		tryLogDiagnosticMessage(
			message := message,
			category := TOF_Core.LOG_CATEGORY.ERROR,
			topic1 := TO_WSTRING(ClassName),
			topic2 := "FileHandleResourceManager.executeRelease",
			topic3 := "FileHandleResourceManager.executeRelease.Done"
		);
	ELSE
		TOF_Core.WideStrings.Append255(
			message,
			"File '",
			TO_WSTRING(_FileOpen.sPathName),
			"' closed");

		tryLogDiagnosticMessage(
			message := message,
			category := TOF_Core.LOG_CATEGORY.INFORMATION,
			topic1 := TO_WSTRING(ClassName),
			topic2 := TO_WSTRING(__POUNAME())
		);
	END_IF

END_IF
END_METHOD


//! <param name="bInCopyCode">
//! if TRUE, the exit method is called for exiting an instance that is copied afterwards (online change).
//! </param>

(*!
<summary>Makes a final best-effort close request for a still-acquired file handle.</summary>
<description>
Does not wait for bBusy to clear or inspect the close result. Callers must complete normal release through
cyclic Execute before destroying this manager; this fallback does not guarantee that the file has closed. Does
not create framework exceptions or format diagnostics. The same fallback runs when bInCopyCode is TRUE; this
method implements no handoff of an active handle to a copied instance. Before online change, callers must
finish normal release and resolve any cleanup error. Under that precondition this fallback has no acquired
handle to close. It cannot prepare an active manager for online change or guarantee uninterrupted file I/O.
</description>
*)
METHOD FB_exit : BOOL
VAR_INPUT
	
	bInCopyCode	: BOOL;
END_VAR
IF _FileHandleAcquired THEN
	_FileClose(hFile := _FileOpen.hFile, bExecute := TRUE);
	_FileOpen(bExecute := FALSE);	
END_IF
END_METHOD

(*!
<summary>Provides the native handle associated with the file resource.</summary>
<description>
Use only during the current acquisition; the value alone is not an acquisition guard. Do not close it
independently or retain it across release.
</description>
*)
{attribute 'monitoring' := 'call'}
PROPERTY FINAL FileHandle : UINT
GET
FileHandle := _FileOpen.hFile;
END_GET
END_PROPERTY

(*!
<summary>Provides the manager-owned typed resource for binding file-content tasks.</summary>
<description>
The reference is valid only while this manager is alive. Obtaining it does not acquire or open a file. It
remains a borrowed view across release and reacquisition; use its handle only during the current acquisition.
Do not delete the resource or modify its borrowed path. No ownership is transferred.
</description>
*)
PROPERTY FileHandleResource : REFERENCE TO FileHandleResource
GET
FileHandleResource REF= _FileHandleResource;
END_GET
END_PROPERTY

(*!
<summary>Provides the configured path for the file operation.</summary>
<description>
Configure before acquisition and keep unchanged through release. Assignment copies the path without opening a
file; StartAcquire rejects a missing path.
</description>
*)
{attribute 'monitoring' := 'call'}
PROPERTY FilePath : Tc2_System.T_MaxString
GET
FilePath := _FileOpen.sPathName;
END_GET
SET
_FileOpen.sPathName := FilePath;
END_SET
END_PROPERTY

(*!
<summary>Finishes a pending open during stopping without starting a new open.</summary>
<description>
TRUE means its response has been processed (or none was pending), and acquisition is no longer scheduled.
Preserve a successfully returned handle so the normal release path can close it.
</description>
*)

METHOD INTERNAL FinishPendingAcquire : BOOL
IF _FileOpen.bBusy THEN
	_FileOpen(bExecute := FALSE);

	IF NOT _FileOpen.bBusy AND_THEN NOT _FileOpen.bError AND_THEN _FileOpen.hFile > 0 THEN
		_FileHandleAcquired := TRUE;
	END_IF
END_IF

FinishPendingAcquire := NOT _FileOpen.bBusy;

IF FinishPendingAcquire THEN
	_Acquiring := FALSE;
END_IF
END_METHOD

(*!
<summary>Returns a borrowed resource object owned by this manager.</summary>
<description>
The caller must not delete the returned object. It may be obtained before acquisition and retained while the
manager remains alive, including across release and reacquisition. The object remains valid after release, but
its presence does not mean the resource is acquired. Use the underlying resource only after successful
acquisition and before release begins. Do not reuse a handle saved from an earlier acquisition after release.
</description>
*)
METHOD GetResource : TOF_Core.IObject
GetResource := _FileHandleResource;
END_METHOD

(*!
<summary>Selects native file access and text or binary flags.</summary>
<description>
Use the valid Tc2_System FOPEN_MODE combinations documented by FileContentManager.ModeFlags. Configure before
acquisition and keep unchanged through release; native opening reports incompatible flags.
</description>
*)

{attribute 'monitoring' := 'call'}

PROPERTY ModeFlags : DWORD
GET
ModeFlags := _FileOpen.nMode;
END_GET
SET
_FileOpen.nMode := ModeFlags;
END_SET
END_PROPERTY

(*!
<summary>Provides the library namespace used in diagnostics.</summary>
<description>Returns borrowed read-only namespace storage; do not modify the referenced string.</description>
*)
{attribute 'monitoring' := 'call'}
PROPERTY NamespaceName : REFERENCE TO STRING
GET
NamespaceName REF= CurrentNamespace.Name;
END_GET
END_PROPERTY

(*!
<summary>Selects the native path context for the filesystem request.</summary>
<description>
Passed to native file opening. Configure before acquisition and keep unchanged through release; the setter
does not validate or open a path.
</description>
*)
{attribute 'monitoring' := 'call'}
PROPERTY PathType : Tc2_System.E_OpenPath
GET
PathType := _FileOpen.ePath;
END_GET
SET
_FileOpen.ePath := PathType;
END_SET
END_PROPERTY

(*!
<summary>Reports whether this manager currently retains an acquired handle.</summary>
<description>
FALSE also occurs before acquisition completes and after a failed best-effort close attempt. This bookkeeping
flag is not proof that the native service physically released a resource.
</description>
*)
{attribute 'monitoring' := 'call'}
PROPERTY ResourceAcquired : BOOL
GET
ResourceAcquired := _FileHandleAcquired;
END_GET
END_PROPERTY

(*!
<summary>Reports the size of this concrete instance in bytes.</summary>
*)
{attribute 'monitoring' := 'call'}
PROPERTY SelfSize : ULINT
GET
SelfSize := XSIZEOF(THIS^);
END_GET
END_PROPERTY

(*!
<summary>Requests opening of the configured file on subsequent Execute calls.</summary>
<description>
Call once with no pending operation. An already acquired handle is retained. An empty FilePath raises an
exception before the request is scheduled. Computed diagnostic strings are held in local buffers for the
duration of the receiving call.
</description>
*)
METHOD StartAcquire
VAR
	formattedLogMessage : WSTRING(255);
END_VAR
IF _FileHandleAcquired THEN
	RETURN;
END_IF

IF TOF_Core.Strings.IsNullOrWhiteSpace(stringToCheck := _FileOpen.sPathName) THEN
	TOF_Core.Exceptions.ThrowDataMemberNotSpecified(
		sourceNamespaceName := NamespaceName,
		sourceClassName := ClassName,
		sourcePOUName := __POUNAME(),
		sourcePosition := __POSITION(),
		dataMemberName := 'FilePath'
	);
END_IF

formattedLogMessage := TOF_Core.WideStrings.Concat255("Attempt to open file '", TO_WSTRING(_FileOpen.sPathName), "'");

tryLogDiagnosticMessage(
	message := formattedLogMessage,
	category := TOF_Core.LOG_CATEGORY.INFORMATION,
	topic1 := TO_WSTRING(ClassName),
	topic2 := TO_WSTRING(__POUNAME())
);

_FileClose(bExecute := FALSE);
_FileOpen(bExecute := FALSE);
_Acquiring := TRUE;
END_METHOD

(*!
<summary>Requests best-effort closing on subsequent Execute calls.</summary>
<description>
Acquisition must have completed or been drained by FinishPendingAcquire. Call once; releasing an absent handle
is allowed. Computed diagnostic strings are held in local buffers for the duration of the receiving call.
</description>
*)
METHOD StartRelease
VAR
	formattedLogMessage : WSTRING(255);
END_VAR
formattedLogMessage := TOF_Core.WideStrings.Concat255("Attempt to close file '", TO_WSTRING(_FileOpen.sPathName), "'");

tryLogDiagnosticMessage(
	message := formattedLogMessage,
	category := TOF_Core.LOG_CATEGORY.INFORMATION,
	topic1 := TO_WSTRING(ClassName),
	topic2 := TO_WSTRING(__POUNAME())
);

IF _FileHandleAcquired THEN
	_Releasing := TRUE;
ELSE
	_FileOpen(bExecute := FALSE);
END_IF
END_METHOD

(*!
<summary>Configures the timeout passed to native operation requests.</summary>
<description>
Shared by native open and close. Configure before acquisition and keep unchanged through release. It is not an
overall resource-lifecycle deadline.
</description>
*)
{attribute 'monitoring' := 'call'}
PROPERTY Timeout : TIME
GET
Timeout := _FileOpen.tTimeout;
END_GET
SET
_FileOpen.tTimeout := Timeout;
_FileClose.tTimeout := Timeout;
END_SET
END_PROPERTY

(*!
<summary>Reports an internal message through the configured diagnostic route.</summary>
<description>
Uses the borrowed DiagnosticLogger directly when present; otherwise retains LogManager topics and routing.
Contains destination exceptions without recursive logging. Returns FALSE on observed terminal allocation
failure; prior diagnostic effects are not rolled back and the fatal latch remains set.
</description>
*)
METHOD PRIVATE tryLogDiagnosticMessage : BOOL
VAR_IN_OUT CONSTANT
	message : TOF_Core.ERROR_MESSAGE;
END_VAR
VAR_INPUT
	category : TOF_Core.LOG_CATEGORY;
	topic1 : WSTRING := "";
	topic2 : WSTRING := "";
	topic3 : WSTRING := "";
END_VAR
__TRY

	IF TOF_Core.DynamicMemoryManager.HasAllocationFailed THEN
		RETURN;
	END_IF

	IF _DiagnosticLogger <> 0 THEN
		tryLogDiagnosticMessage := _DiagnosticLogger.TryLogMessage(category := category, message := message);
	ELSE
		tryLogDiagnosticMessage := TOF_Core.LogManager.TryLogMessage(
			category := category,
			message := message,
			topic1 := topic1,
			topic2 := topic2,
			topic3 := topic3
		);
	END_IF

	IF TOF_Core.DynamicMemoryManager.HasAllocationFailed THEN
		tryLogDiagnosticMessage := FALSE;
	END_IF

__CATCH
	// Diagnostic failure must not replace the task lifecycle outcome.
	tryLogDiagnosticMessage := FALSE;
__ENDTRY
END_METHOD

END_FUNCTION_BLOCK

// ---- Tasks/File/FileContent/FileHandleResource.TcPOU
(*
SPDX-FileCopyrightText: © 2026 Oleksandr Tiutyk <trofimich@gmail.com>
SPDX-License-Identifier: MIT
License: https://opensource.org/license/mit
*)

(*!
<summary>Exposes a borrowed view of the native open-file block owned by a resource manager.</summary>
<description>
This object owns neither the native block nor its handle. Keep the referenced FB_FileOpen alive for the entire
use of this view. The getters do not check acquisition: an assigned view is not evidence of an open file. Use
handle and target together only during the current acquisition, never after release. An invalid native-block
reference yields default scalar results or an invalid FilePath reference. Do not modify FilePath through its
reference, close the handle independently or delete this borrowed object.
</description>
*)

{attribute 'no_explicit_call' := 'Direct call is not allowed'}
FUNCTION_BLOCK INTERNAL FileHandleResource EXTENDS TOF_Core.Object
VAR_STAT
	//! <summary>Class name shared by all instances of this function block.</summary>
	{attribute 'hide'} 
	_ClassName : STRING := __POUNAME();
END_VAR
VAR
	{attribute 'hide'} 
	_FileOpen : REFERENCE TO Tc2_System.FB_FileOpen;
END_VAR

(*!
<summary>Target of the open file; use together with FileHandle.</summary>
*)

{attribute 'monitoring' := 'call'}

PROPERTY AmsNetId : Tc2_System.T_AmsNetID
GET
IF __ISVALIDREF(_FileOpen) THEN
	AmsNetId := _FileOpen.sNetId;
END_IF
END_GET
END_PROPERTY

(*!
<summary>Provides the concrete type name used in diagnostics.</summary>
<description>
Returns borrowed read-only metadata; keep the instance alive and do not modify the referenced string.
Reading does not allocate memory, initialize resources or transfer ownership.
</description>
*)
{attribute 'monitoring' := 'call'}
PROPERTY ClassName : REFERENCE TO STRING
GET
ClassName REF= _ClassName;
END_GET
END_PROPERTY

(*!
<summary>Binds this view to a caller-owned native file-open block without acquiring a file.</summary>
<description>
The binding is borrowed and must remain alive throughout use. An invalid reference is retained without
throwing; getters then return default scalars or an invalid reference. No handle is opened or closed.
</description>
<param name="fileOpen">Borrowed native block providing the path, target and current handle.</param>
*)
METHOD FB_Init: BOOL
VAR_INPUT
	bInitRetains : BOOL; // TRUE: the retain variables are initialized (reset warm / reset cold)
	bInCopyCode : BOOL;  // TRUE: the instance will be copied to the copy code afterward (online change)
	fileOpen : REFERENCE TO Tc2_System.FB_FileOpen;
END_VAR
_FileOpen REF= fileOpen;
END_METHOD

(*!
<summary>Reads the native handle from the borrowed open-file block.</summary>
<description>
Returns the default UINT when no native block is bound. Does not check acquisition or close status; a stored
numeric handle must not be reused after release.
</description>
*)
{attribute 'monitoring' := 'call'}
PROPERTY FileHandle : UINT
GET
IF __ISVALIDREF(_FileOpen) THEN
	FileHandle := _FileOpen.hFile;
END_IF
END_GET
END_PROPERTY

(*!
<summary>Provides a borrowed view of the configured native file path.</summary>
<description>
The reference is invalid when no native block is bound. Keep the owner alive and do not write through this
reference. This path identifies configuration, not proof that the file is open.
</description>
*)
{attribute 'monitoring' := 'call'}
PROPERTY FilePath : REFERENCE TO Tc2_System.T_MaxString
GET
IF __ISVALIDREF(_FileOpen) THEN
	FilePath REF= _FileOpen.sPathName;
END_IF
END_GET
END_PROPERTY

(*!
<summary>Provides the library namespace used in diagnostics.</summary>
<description>Returns borrowed read-only namespace storage; do not modify the referenced string.</description>
*)
{attribute 'monitoring' := 'call'}
PROPERTY NamespaceName : REFERENCE TO STRING
GET
NamespaceName REF= CurrentNamespace.Name;
END_GET
END_PROPERTY

(*!
<summary>Reports the size of this concrete instance in bytes.</summary>
*)
{attribute 'monitoring' := 'call'}
PROPERTY SelfSize : ULINT
GET
SelfSize := XSIZEOF(THIS^);
END_GET
END_PROPERTY

END_FUNCTION_BLOCK

// ---- Tasks/File/FileContent/Tasks/CheckEndOfFile.TcPOU
(*
SPDX-FileCopyrightText: © 2026 Oleksandr Tiutyk <trofimich@gmail.com>
SPDX-License-Identifier: MIT
License: https://opensource.org/license/mit
*)

(*!
<summary>Queries the native end-of-file status of the acquired file.</summary>
<description>
The owner must keep the resource acquired through stopping. Configure Timeout before Start and keep it
unchanged until STOPPED. Missing binding and native errors use the Task failure and cleanup path. IsEndOfFile
exposes the native result only after STOPPED with WORK_DONE; FALSE outside that state does not establish that
more data is available. Cancellation waits for a submitted query. Reset clears binding and request state while
retaining Timeout.
</description>
*)

{attribute 'no_explicit_call' := 'do not call this function block directly'}
FUNCTION_BLOCK CheckEndOfFile EXTENDS FileContentTask
VAR_STAT
	//! <summary>Static type metadata available before the base task initializes its default name.</summary>
	{attribute 'hide'}
	_ClassName : STRING := __POUNAME();
END_VAR
VAR
    _CheckEOF : Tc2_System.FB_EOF;
END_VAR

(*!
<summary>Exposes the native operation target copied from the bound file resource.</summary>
<description>
The resource target overwrites a separately assigned value before native submission. Configure the resource
owner to select a target; do not change this value while the task is running.
</description>
*)
{attribute 'monitoring' := 'call'}
PROPERTY AmsNetId : Tc2_System.T_AmsNetID
GET
AmsNetId := _CheckEOF.sNetId;
END_GET
SET
_CheckEOF.sNetId := AmsNetId;
END_SET
END_PROPERTY

(*!
<summary>Provides the concrete type name used in diagnostics.</summary>
<description>
Returns borrowed read-only metadata; keep the instance alive and do not modify the referenced string.
Initialized static storage is ready during base Task.FB_init; this getter has no side effects or exceptions.
</description>
*)
{attribute 'monitoring' := 'call'}
PROPERTY ClassName : REFERENCE TO STRING
GET
ClassName REF= _ClassName;
END_GET
END_PROPERTY

(*!
<summary>Reports whether the underlying native file operation is busy.</summary>
<description>
Observes native I/O, including work drained during stopping. FALSE is not a task-success result and does not
independently permit the resource owner to close or destroy the file.
</description>
*)
{attribute 'monitoring' := 'call'}
PROPERTY FileOperationInProgress : BOOL
GET
FileOperationInProgress := _CheckEOF.bBusy;
END_GET
END_PROPERTY

(*!
<summary>Reports the EOF indicator obtained by a successfully completed check.</summary>
<description>
Returns the native result only while State.Stopped and FinalStopReason.WorkDone are both TRUE. In every other
state, including READY, RUNNING, failure and cancellation, returns the initial value of the property type.
This default is not a success indicator; inspect the task state and final reason. FALSE outside successful
completion does not establish that more data is available. The getter does not modify native outputs or
buffers. Copy a successful result before Reset or reuse.
</description>
*)
{attribute 'monitoring' := 'call'}
PROPERTY IsEndOfFile : BOOL
GET
IF NOT State.Stopped OR_ELSE NOT FinalStopReason.WorkDone THEN
	RETURN;
END_IF

IsEndOfFile := _CheckEOF.bEOF;
END_GET
END_PROPERTY

(*!
<summary>Provides the library namespace used in diagnostics.</summary>
<description>Returns borrowed read-only namespace storage; do not modify the referenced string.</description>
*)
{attribute 'monitoring' := 'call'}
PROPERTY NamespaceName : REFERENCE TO STRING
GET
NamespaceName REF= CurrentNamespace.Name;
END_GET
END_PROPERTY

(*!
<summary>Resets the native request edge after the task has stopped.</summary>
<description>
Also preserves the inherited resource-binding cleanup. Configured inputs remain available for reuse; borrowed
buffers are not freed or cleared. Pending I/O must finish during stopping before this hook runs.
</description>
*)
METHOD PROTECTED OnReset
SUPER^.OnReset();

_CheckEOF(bExecute := FALSE);
END_METHOD

(*!
<summary>Checks the end-of-file indicator through the bound file handle.</summary>
<description>
Requires a live bound resource whose owner keeps the handle acquired until stopping completes. Native errors
raise an exception for the base Task failure and cleanup path without dynamic string-builder allocations;
completed I/O effects are not rolled back.
</description>
<param name="processingState">BUSY while pending; DONE after native completion without an error.</param>
<param name="stopReasonMessage">Not changed; native failures use exceptions.</param>
*)
METHOD PROTECTED OnRunning
VAR_OUTPUT
	processingState : TOF_Tasks.TASK_PROCESSING_STATE;
END_VAR
VAR_IN_OUT
	stopReasonMessage : TOF_Core.ERROR_MESSAGE;
END_VAR
VAR
	errorMessage : TOF_Core.ERROR_MESSAGE;
END_VAR
IF NOT _CheckEOF.bExecute THEN 
	IF NOT __ISVALIDREF(_FileHandleResource) THEN
		TOF_Core.Exceptions.ThrowDataMemberNotSpecified(
			sourceNamespaceName := NamespaceName,
			sourceClassName := ClassName,
			sourcePOUName := __POUNAME(),
			sourcePosition := __POSITION(),
			dataMemberName := 'FileHandleResource'
		);		
	END_IF
	
	_CheckEOF.sNetId := _FileHandleResource.AmsNetId;
	_CheckEOF.hFile := _FileHandleResource.FileHandle;
END_IF

_CheckEOF(bExecute := TRUE);

IF _CheckEOF.bError THEN
	TOF_Core.WideStrings.Append255(
		errorMessage,
		"An error occurred while checking end of file '",
		TO_WSTRING(FilePath),
		"'");

	FileSystemExceptions.ThrowFileSystem(
		sourceNamespaceName := NamespaceName,
		sourceClassName := ClassName,
		sourcePOUName := __POUNAME(),
		sourcePosition := __POSITION(),
		message := errorMessage,
		errorCode := _CheckEOF.nErrId
	);
END_IF

IF NOT _CheckEOF.bBusy THEN
	processingState := TOF_Tasks.TASK_PROCESSING_STATE.DONE;
END_IF
END_METHOD

(*!
<summary>Wait for an already submitted file operation before allowing handle release.</summary>
<description>
FALSE on bExecute only avoids a new request; it does not abort the pending one. Runs for every stop reason. If
no operation is busy, stopping is ready immediately.
</description>
<param name="readyToRelease">TRUE after pending work has completed and release may begin.</param>
*)

METHOD PROTECTED OnStopping
VAR_OUTPUT
	readyToRelease : BOOL;
END_VAR
IF _CheckEOF.bBusy THEN
	_CheckEOF(bExecute := FALSE);
END_IF

readyToRelease := NOT _CheckEOF.bBusy;
END_METHOD

(*!
<summary>Reports the size of this concrete instance in bytes.</summary>
*)
{attribute 'monitoring' := 'call'}
PROPERTY SelfSize : ULINT
GET
SelfSize := XSIZEOF(THIS^);
END_GET
END_PROPERTY

(*!
<summary>Configures the timeout passed to native operation requests.</summary>
<description>
Set before Start and keep unchanged until STOPPED. Reset preserves this value. It is not an overall task
deadline or a guarantee of resource release after a timeout.
</description>
*)
{attribute 'monitoring' := 'call'}
PROPERTY Timeout : TIME
GET
Timeout := _CheckEOF.tTimeout;
END_GET
SET
_CheckEOF.tTimeout := Timeout;
END_SET
END_PROPERTY

END_FUNCTION_BLOCK

// ---- Tasks/File/FileContent/Tasks/FileContentTask.TcPOU
(*
SPDX-FileCopyrightText: © 2026 Oleksandr Tiutyk <trofimich@gmail.com>
SPDX-License-Identifier: MIT
License: https://opensource.org/license/mit
*)

(*!
<summary>Base for a file-content operation borrowing a manager-owned file resource.</summary>
<description>
Queue membership and resource binding do not transfer ownership. One owner drives the task. Keep the resource
owner alive while using its binding; an assigned reference alone does not prove acquisition. The manager
acquires the file before child execution and waits for child stopping before release. Removing a child from a
queue does not clear the binding. Reset from STOPPED clears it; READY Reset is a no-op. A removed READY child
must explicitly clear or replace its binding before the old owner is destroyed. Descendants overriding OnReset
must preserve binding cleanup. Descendants must finish native pending I/O during stopping before allowing the
parent to release the resource. Do not mutate borrowed resource data.
</description>
*)

FUNCTION_BLOCK ABSTRACT FileContentTask EXTENDS TOF_Tasks.Task IMPLEMENTS IFileContentTask
VAR
	_FileHandleResource : REFERENCE TO FileHandleResource;
END_VAR

(*!
<summary>File-content operations take the actual target from the bound resource</summary>
<description>
before submitting I/O, overriding any separately configured AmsNetId.
</description>
*)

{attribute 'monitoring' := 'call'}

PROPERTY ABSTRACT AmsNetId : Tc2_System.T_AmsNetID
GET
END_GET
SET
END_SET
END_PROPERTY

(*!
<summary>Reads the handle through the current borrowed resource binding.</summary>
<description>
Returns the default UINT when unbound. Does not establish acquisition; use only while the owning manager has
acquired the current file, and do not cache across release.
</description>
*)
{attribute 'monitoring' := 'call'}
PROPERTY FINAL FileHandle : UINT
GET
IF __ISVALIDREF(_FileHandleResource) THEN
	FileHandle := _FileHandleResource.FileHandle;
END_IF
END_GET
END_PROPERTY

(*!
<summary>Exposes the borrowed resource binding for this operation.</summary>
<description>
Returns an invalid reference when unbound. The owner must remain alive throughout access; an assigned
reference does not mean the file is acquired. Do not mutate borrowed data or close the handle independently.
</description>
*)
{attribute 'monitoring' := 'call'}
PROPERTY FINAL FileHandleResource : REFERENCE TO FileHandleResource
GET
IF __ISVALIDREF(_FileHandleResource) THEN
	FileHandleResource REF= _FileHandleResource;
END_IF
END_GET
END_PROPERTY

(*!
<summary>Copies the file path from the current resource binding.</summary>
<description>
Returns the default empty string when unbound. Reading requires the resource owner to remain alive; the path
is configuration and does not prove acquisition.
</description>
*)
{attribute 'monitoring' := 'call'}
PROPERTY FINAL FilePath : Tc2_System.T_MaxString
GET
IF __ISVALIDREF(_FileHandleResource) THEN
	FilePath := _FileHandleResource.FilePath;
END_IF
END_GET
END_PROPERTY

(*!
<summary>Clears the borrowed resource binding when a STOPPED child is reset.</summary>
<description>
Base Reset does not call this hook in READY. Overriding descendants must preserve this cleanup; it neither
closes the file nor removes the task from any queue.
</description>
*)
METHOD PROTECTED OnReset
_FileHandleResource REF= 0;
END_METHOD

(*!
<summary>Bind, replace or clear a borrowed resource only in READY; otherwise throw.</summary>
<description>
An invalid reference clears the binding. Reset a STOPPED task before rebinding. The caller must first remove
the task from any queue; READY alone does not mean it is unqueued. The resource owner must outlive its use by
this task. Queue removal does not clear this binding; READY Reset is a no-op. Clear or replace the binding
explicitly for a removed READY task before destroying the old resource owner.
</description>
*)

METHOD SetFileHandleResource
VAR_INPUT
	fileHandleResource : REFERENCE TO FileHandleResource;
END_VAR
IF NOT State.Ready THEN
	TOF_Core.Exceptions.ThrowStandard(
		sourceNamespaceName := NamespaceName,
		sourceClassName := ClassName,
		sourcePOUName := __POUNAME(),
		sourcePosition := __POSITION(),
		message := "FileHandleResource can only be assigned in READY state"
	);
END_IF

IF __ISVALIDREF(fileHandleResource) THEN
	_FileHandleResource REF= fileHandleResource;
ELSE
	_FileHandleResource REF= 0;
END_IF
END_METHOD

(*!
<summary>Configures the timeout passed to native operation requests.</summary>
<description>
Implementations apply this value to their native requests. Configure before execution and keep stable through
stopping; it is not a deadline for the entire task lifecycle.
</description>
*)
{attribute 'monitoring' := 'call'}
{attribute 'OPC.UA.DA.Property' := '1'}
{attribute 'OPC.UA.DA' := '1'}
PROPERTY ABSTRACT Timeout : TIME
GET
END_GET
SET
END_SET
END_PROPERTY

(*!
<summary>TRUE while the underlying file FB reports a pending request, including</summary>
<description>
cancellation wait. Reading has no side effects and does not indicate task lifecycle state or permission to
release the file resource.
</description>
*)

{attribute 'monitoring' := 'call'}

PROPERTY ABSTRACT FileOperationInProgress : BOOL
GET
END_GET
END_PROPERTY

END_FUNCTION_BLOCK

// ---- Tasks/File/FileContent/Tasks/SetPositionInFile.TcPOU
(*
SPDX-FileCopyrightText: © 2026 Oleksandr Tiutyk <trofimich@gmail.com>
SPDX-License-Identifier: MIT
License: https://opensource.org/license/mit
*)

(*!
<summary>Changes the bound file's position using a configured offset and origin.</summary>
<description>
The resource owner must keep the file acquired through task stopping. Configure Position, Origin and Timeout
before Start and keep them unchanged until STOPPED. Missing binding and native errors use the base Task
failure and cleanup path. Cancellation waits for submitted I/O and does not restore the previous file
position. Reset from STOPPED clears the binding and native request state, preserving offset, origin and
timeout.
</description>
*)

{attribute 'no_explicit_call' := 'do not call this function block directly'}
FUNCTION_BLOCK SetPositionInFile EXTENDS FileContentTask
VAR_STAT
	//! <summary>Static type metadata available before the base task initializes its default name.</summary>
	{attribute 'hide'}
	_ClassName : STRING := __POUNAME();
END_VAR
VAR
    _SetPosition : Tc2_System.FB_FileSeek;
END_VAR

(*!
<summary>Exposes the native operation target copied from the bound file resource.</summary>
<description>
The resource target overwrites a separately assigned value before native submission. Configure the resource
owner to select a target; do not change this value while the task is running.
</description>
*)
{attribute 'monitoring' := 'call'}
PROPERTY AmsNetId : Tc2_System.T_AmsNetID
GET
AmsNetId := _SetPosition.sNetId;
END_GET
SET
_SetPosition.sNetId := AmsNetId;
END_SET
END_PROPERTY

(*!
<summary>Provides the concrete type name used in diagnostics.</summary>
<description>
Returns borrowed read-only metadata; keep the instance alive and do not modify the referenced string.
Initialized static storage is ready during base Task.FB_init; this getter has no side effects or exceptions.
</description>
*)
{attribute 'monitoring' := 'call'}
PROPERTY ClassName : REFERENCE TO STRING
GET
ClassName REF= _ClassName;
END_GET
END_PROPERTY

(*!
<summary>Reports whether the underlying native file operation is busy.</summary>
<description>
Observes native I/O, including work drained during stopping. FALSE is not a task-success result and does not
independently permit the resource owner to close or destroy the file.
</description>
*)
{attribute 'monitoring' := 'call'}
PROPERTY FileOperationInProgress : BOOL
GET
FileOperationInProgress := _SetPosition.bBusy;
END_GET
END_PROPERTY

(*!
<summary>Provides the library namespace used in diagnostics.</summary>
<description>Returns borrowed read-only namespace storage; do not modify the referenced string.</description>
*)
{attribute 'monitoring' := 'call'}
PROPERTY NamespaceName : REFERENCE TO STRING
GET
NamespaceName REF= CurrentNamespace.Name;
END_GET
END_PROPERTY

(*!
<summary>Clears the borrowed binding and native request state after stopping.</summary>
<description>
Preserves Position, Origin and Timeout. Does not cancel pending I/O; stopping must finish first.
</description>
*)
METHOD PROTECTED OnReset
SUPER^.OnReset();

_SetPosition(bExecute := FALSE);
END_METHOD

(*!
<summary>Changes the position of the bound file using the configured offset and origin.</summary>
<description>
Requires a live bound resource whose owner keeps the handle acquired until stopping completes. Native errors
raise an exception for the base Task failure and cleanup path without dynamic string-builder allocations;
completed I/O effects are not rolled back.
</description>
<param name="processingState">BUSY while pending; DONE after native completion without an error.</param>
<param name="stopReasonMessage">Not changed; native failures use exceptions.</param>
*)
METHOD PROTECTED OnRunning
VAR_OUTPUT
	processingState : TOF_Tasks.TASK_PROCESSING_STATE;
END_VAR
VAR_IN_OUT
	stopReasonMessage : TOF_Core.ERROR_MESSAGE;
END_VAR
VAR
	errorMessage : TOF_Core.ERROR_MESSAGE;
END_VAR
IF NOT _SetPosition.bExecute THEN 
	IF NOT __ISVALIDREF(_FileHandleResource) THEN
		TOF_Core.Exceptions.ThrowDataMemberNotSpecified(
			sourceNamespaceName := NamespaceName,
			sourceClassName := ClassName,
			sourcePOUName := __POUNAME(),
			sourcePosition := __POSITION(),
			dataMemberName := 'FileHandleResource'
		);		
	END_IF
	
	_SetPosition.sNetId := _FileHandleResource.AmsNetId;
	_SetPosition.hFile := _FileHandleResource.FileHandle;
END_IF

_SetPosition(bExecute := TRUE);

IF _SetPosition.bError THEN
	TOF_Core.WideStrings.Append255(
		errorMessage,
		"An error occurred while changing position in file ",
		TO_WSTRING(FilePath),
		"'");

	FileSystemExceptions.ThrowFileSystem(
		sourceNamespaceName := NamespaceName,
		sourceClassName := ClassName,
		sourcePOUName := __POUNAME(),
		sourcePosition := __POSITION(),
		message := errorMessage,
		errorCode := _SetPosition.nErrId
	);
END_IF

IF NOT _SetPosition.bBusy THEN
	processingState := TOF_Tasks.TASK_PROCESSING_STATE.DONE;
END_IF
END_METHOD

(*!
<summary>Wait for an already submitted file operation before allowing handle release.</summary>
<description>
FALSE on bExecute only avoids a new request; it does not abort the pending one. Runs for every stop reason. If
no operation is busy, stopping is ready immediately.
</description>
<param name="readyToRelease">TRUE after pending work has completed and release may begin.</param>
*)

METHOD PROTECTED OnStopping
VAR_OUTPUT
	readyToRelease : BOOL;
END_VAR
IF _SetPosition.bBusy THEN
	_SetPosition(bExecute := FALSE);
END_IF

readyToRelease := NOT _SetPosition.bBusy;
END_METHOD

{attribute 'monitoring' := 'call'}
(*!
<summary>Selects the native reference point for the requested offset.</summary>
<description>
Configure together with Position before Start and keep unchanged until STOPPED. Passed to FB_FileSeek without
additional validation; Reset preserves it.
</description>
*)
PROPERTY Origin : Tc2_System.E_SeekOrigin
GET
Origin := _SetPosition.eOrigin;
END_GET
SET
_SetPosition.eOrigin := Origin;
END_SET
END_PROPERTY

{attribute 'monitoring' := 'call'}
(*!
<summary>Provides the requested native seek offset relative to Origin.</summary>
<description>
This is configuration, not the resulting file position. Set before Start and keep unchanged until STOPPED;
Reset preserves it. Native constraints depend on Origin and the opened file.
</description>
*)
PROPERTY Position : DINT
GET
Position := _SetPosition.nSeekPos;
END_GET
SET
_SetPosition.nSeekPos := Position;
END_SET
END_PROPERTY

(*!
<summary>Reports the size of this concrete instance in bytes.</summary>
*)
{attribute 'monitoring' := 'call'}
PROPERTY SelfSize : ULINT
GET
SelfSize := XSIZEOF(THIS^);
END_GET
END_PROPERTY

(*!
<summary>Configures the timeout passed to native operation requests.</summary>
<description>
Set before Start and keep unchanged until STOPPED. Reset preserves this value. It is not an overall task
deadline or a guarantee of resource release after a timeout.
</description>
*)
{attribute 'monitoring' := 'call'}
PROPERTY Timeout : TIME
GET
Timeout := _SetPosition.tTimeout;
END_GET
SET
_SetPosition.tTimeout := Timeout;
END_SET
END_PROPERTY

END_FUNCTION_BLOCK

// ---- Tasks/File/FileContent/Tasks/WriteBytesToFile.TcPOU
(*
SPDX-FileCopyrightText: © 2026 Oleksandr Tiutyk <trofimich@gmail.com>
SPDX-License-Identifier: MIT
License: https://opensource.org/license/mit
*)

(*!
<summary>Performs a cyclic file byte transfer through a borrowed file resource.</summary>
<description>
Configure SourceBuffer and BytesCountToWrite before Start and keep them stable until STOPPED. The caller owns
the buffer and must keep at least the requested number of bytes readable and unchanged through stopping. A
null buffer or zero count raises DataMemberNotSpecifiedException before the native request; the base Task
records FAILURE and completes its cleanup. Buffer capacity and the validity of non-null addresses are caller
preconditions, not checked here. No ownership is transferred and partial I/O effects are not rolled back.
</description>
*)

{attribute 'no_explicit_call' := 'do not call this function block directly'}
FUNCTION_BLOCK WriteBytesToFile EXTENDS FileContentTask
VAR_STAT
	//! <summary>Static type metadata available before the base task initializes its default name.</summary>
	{attribute 'hide'}
	_ClassName : STRING := __POUNAME();
END_VAR
VAR
    _WriteBytes : Tc2_System.FB_FileWrite;
END_VAR

(*!
<summary>Reports the byte count from a successfully completed write.</summary>
<description>
Returns the native result only while State.Stopped and FinalStopReason.WorkDone are both TRUE. In every other
state, including READY, RUNNING, failure and cancellation, returns the initial value of the property type.
This default is not a success indicator; inspect the task state and final reason. Zero after failure or
cancellation does not mean no bytes were written; partial native effects are not rolled back. The getter does
not modify native outputs or buffers. Copy a successful result before Reset or reuse.
</description>
*)
{attribute 'monitoring' := 'call'}
PROPERTY ActuallyWrittenBytes : UDINT
GET
IF NOT State.Stopped OR_ELSE NOT FinalStopReason.WorkDone THEN
	RETURN;
END_IF

ActuallyWrittenBytes := _WriteBytes.cbWrite;
END_GET
END_PROPERTY

(*!
<summary>Exposes the native operation target copied from the bound file resource.</summary>
<description>
The resource target overwrites a separately assigned value before native submission. Configure the resource
owner to select a target; do not change this value while the task is running.
</description>
*)
{attribute 'monitoring' := 'call'}
PROPERTY AmsNetId : Tc2_System.T_AmsNetID
GET
AmsNetId := _WriteBytes.sNetId;
END_GET
SET
_WriteBytes.sNetId := AmsNetId;
END_SET
END_PROPERTY

(*!
<summary>Specifies the requested byte count.</summary>
<description>
Must be positive and no greater than the available buffer capacity. Zero is rejected by OnRunning before the
native request and results in Task FAILURE after cleanup. The setter stores configuration without validation;
keep the count stable from Start until STOPPED.
</description>
*)
{attribute 'monitoring' := 'call'}
PROPERTY BytesCountToWrite : UDINT
GET
BytesCountToWrite := _WriteBytes.cbWriteLen;
END_GET
SET
_WriteBytes.cbWriteLen := BytesCountToWrite;
END_SET
END_PROPERTY

(*!
<summary>Provides the concrete type name used in diagnostics.</summary>
<description>
Returns borrowed read-only metadata; keep the instance alive and do not modify the referenced string.
Initialized static storage is ready during base Task.FB_init; this getter has no side effects or exceptions.
</description>
*)
{attribute 'monitoring' := 'call'}
PROPERTY ClassName : REFERENCE TO STRING
GET
ClassName REF= _ClassName;
END_GET
END_PROPERTY

(*!
<summary>Reports whether the underlying native file operation is busy.</summary>
<description>
Observes native I/O, including work drained during stopping. FALSE is not a task-success result and does not
independently permit the resource owner to close or destroy the file.
</description>
*)
{attribute 'monitoring' := 'call'}
PROPERTY FileOperationInProgress : BOOL
GET
FileOperationInProgress := _WriteBytes.bBusy;
END_GET
END_PROPERTY

(*!
<summary>Provides the library namespace used in diagnostics.</summary>
<description>Returns borrowed read-only namespace storage; do not modify the referenced string.</description>
*)
{attribute 'monitoring' := 'call'}
PROPERTY NamespaceName : REFERENCE TO STRING
GET
NamespaceName REF= CurrentNamespace.Name;
END_GET
END_PROPERTY

(*!
<summary>Resets the native request edge after the task has stopped.</summary>
<description>
Also preserves the inherited resource-binding cleanup. Configured inputs remain available for reuse; borrowed
buffers are not freed or cleared. Pending I/O must finish during stopping before this hook runs.
</description>
*)
METHOD PROTECTED OnReset
SUPER^.OnReset();

_WriteBytes(bExecute := FALSE);
END_METHOD

(*!
<summary>Writes the configured byte buffer to the bound file and checks the written count.</summary>
<description>
Requires a live bound resource whose owner keeps the handle acquired until stopping completes. Before
submitting I/O, a null buffer or zero count raises DataMemberNotSpecifiedException for the missing property.
This rejects invalid configuration through the base Task failure and cleanup path. Native errors also raise an
exception without dynamic string-builder allocations; completed I/O effects are not rolled back.
</description>
<param name="processingState">BUSY while pending; DONE after a full write; ERROR on a short write.</param>
<param name="stopReasonMessage">
Receives byte-count diagnostics on a short write; native failures use exceptions.
</param>
*)
METHOD PROTECTED OnRunning
VAR_OUTPUT
	processingState : TOF_Tasks.TASK_PROCESSING_STATE;
END_VAR
VAR_IN_OUT
	stopReasonMessage : TOF_Core.ERROR_MESSAGE;
END_VAR
VAR
	errorMessage : TOF_Core.ERROR_MESSAGE;
END_VAR
IF NOT _WriteBytes.bExecute THEN 
	IF NOT __ISVALIDREF(_FileHandleResource) THEN
		TOF_Core.Exceptions.ThrowDataMemberNotSpecified(
			sourceNamespaceName := NamespaceName,
			sourceClassName := ClassName,
			sourcePOUName := __POUNAME(),
			sourcePosition := __POSITION(),
			dataMemberName := 'FileHandleResource'
		);		
	END_IF
	
	IF _WriteBytes.pWriteBuff = TOF_Core.Memory.NULL_ADDRESS THEN
		TOF_Core.Exceptions.ThrowDataMemberNotSpecified(
			sourceNamespaceName := NamespaceName,
			sourceClassName := ClassName,
			sourcePOUName := __POUNAME(),
			sourcePosition := __POSITION(),
			dataMemberName := 'SourceBuffer'
		);
	END_IF

	IF _WriteBytes.cbWriteLen = TOF_Core.UnsignedInt32.ZERO THEN
		TOF_Core.Exceptions.ThrowDataMemberNotSpecified(
			sourceNamespaceName := NamespaceName,
			sourceClassName := ClassName,
			sourcePOUName := __POUNAME(),
			sourcePosition := __POSITION(),
			dataMemberName := 'BytesCountToWrite'
		);
	END_IF

	_WriteBytes.sNetId := _FileHandleResource.AmsNetId;
	_WriteBytes.hFile := _FileHandleResource.FileHandle;
END_IF

_WriteBytes(bExecute := TRUE);

IF _WriteBytes.bError THEN
	TOF_Core.WideStrings.Append255(
		errorMessage,
		"An error occurred while writing bytes to file ",
		TO_WSTRING(FilePath),
		"'");

	FileSystemExceptions.ThrowFileSystem(
		sourceNamespaceName := NamespaceName,
		sourceClassName := ClassName,
		sourcePOUName := __POUNAME(),
		sourcePosition := __POSITION(),
		message := errorMessage,
		errorCode := _WriteBytes.nErrId
	);
END_IF

IF NOT _WriteBytes.bBusy THEN
	(* A short write may leave bError=FALSE; success requires the full byte count. *)
	IF _WriteBytes.cbWrite <> _WriteBytes.cbWriteLen THEN
		stopReasonMessage := TOF_Core.WideStrings.Concat255(
			"File write byte count mismatch: expected ",
			TO_WSTRING(_WriteBytes.cbWriteLen),
			", written ",
			TO_WSTRING(_WriteBytes.cbWrite)
		);
		
		processingState := TOF_Tasks.TASK_PROCESSING_STATE.ERROR;
	ELSE
		processingState := TOF_Tasks.TASK_PROCESSING_STATE.DONE;
	END_IF
END_IF
END_METHOD

(*!
<summary>Wait for an already submitted file operation before allowing handle release.</summary>
<description>
FALSE on bExecute only avoids a new request; it does not abort the pending one. Runs for every stop reason. If
no operation is busy, stopping is ready immediately.
</description>
<param name="readyToRelease">TRUE after pending work has completed and release may begin.</param>
*)

METHOD PROTECTED OnStopping
VAR_OUTPUT
	readyToRelease : BOOL;
END_VAR
IF _WriteBytes.bBusy THEN
	_WriteBytes(bExecute := FALSE);
END_IF

readyToRelease := NOT _WriteBytes.bBusy;
END_METHOD

(*!
<summary>Reports the size of this concrete instance in bytes.</summary>
*)
{attribute 'monitoring' := 'call'}
PROPERTY SelfSize : ULINT
GET
SelfSize := XSIZEOF(THIS^);
END_GET
END_PROPERTY

(*!
<summary>Provides the caller-owned buffer address for the transfer.</summary>
<description>
Must be non-null before I/O. The caller provides at least BytesCountToWrite bytes of readable and unchanged
storage and retains it until STOPPED, including cancellation cleanup. The setter stores the address without
validating capacity or lifetime; a null address is rejected by OnRunning before the native request. Keep this
setting stable during the run.
</description>
*)
{attribute 'monitoring' := 'call'}
PROPERTY SourceBuffer : PVOID
GET
SourceBuffer := _WriteBytes.pWriteBuff;
END_GET
SET
_WriteBytes.pWriteBuff := SourceBuffer;
END_SET
END_PROPERTY

(*!
<summary>Configures the timeout passed to native operation requests.</summary>
<description>
Set before Start and keep unchanged until STOPPED. Reset preserves this value. It is not an overall task
deadline or a guarantee of resource release after a timeout.
</description>
*)
{attribute 'monitoring' := 'call'}
PROPERTY Timeout : TIME
GET
Timeout := _WriteBytes.tTimeout;
END_GET
SET
_WriteBytes.tTimeout := Timeout;
END_SET
END_PROPERTY

END_FUNCTION_BLOCK

// ---- Tasks/File/LoadFile.TcPOU
(*
SPDX-FileCopyrightText: © 2026 Oleksandr Tiutyk <trofimich@gmail.com>
SPDX-License-Identifier: MIT
License: https://opensource.org/license/mit
*)

(*!
<summary>Loads file contents through cyclic task execution.</summary>
<description>
The native FB_FileLoad opens the file in binary mode, reads the requested byte count and closes it. Its
documented path support is the addressed target's local filesystem, not a network-share path. Use one owner
task. Configure FilePath, AmsNetId, TargetBuffer, TargetBufferSize and Timeout before Start and keep them
unchanged until STOPPED. The caller supplies live writable memory of at least TargetBufferSize bytes and
retains it through stopping after failure or cancellation. Do not access that memory concurrently with the
operation. Missing path, null buffer and zero size are rejected during execution; capacity and pointer
lifetime cannot be verified by this wrapper. Native errors use Task failure handling. Continue Execute until
STOPPED. Cancellation drains pending work without restoring buffer contents. WORK_DONE means the native
request completed without an error; this wrapper does not compare the returned byte count with file size or
promise a complete snapshot of a concurrently modified file. LoadedBytesCount exposes the result only after
STOPPED and WORK_DONE. Reset preserves configuration.
</description>
*)

{attribute 'no_explicit_call' := 'do not call this function block directly'}
FUNCTION_BLOCK LoadFile EXTENDS TOF_Tasks.Task IMPLEMENTS IFileSystemTask
VAR_STAT
	//! <summary>Static type metadata available before the base task initializes its default name.</summary>
	{attribute 'hide'}
	_ClassName : STRING := __POUNAME();
END_VAR
VAR
    _LoadFile : Tc2_System.FB_FileLoad; 
END_VAR

(*!
<summary>Selects the ADS target for the native filesystem operation.</summary>
<description>
Configure before Start and keep unchanged until STOPPED; the setter stores configuration without submitting
I/O.
</description>
*)
{attribute 'monitoring' := 'call'}
PROPERTY AmsNetId : Tc2_System.T_AmsNetID
GET
AmsNetId := _LoadFile.sNetId;
END_GET
SET
_LoadFile.sNetId := AmsNetId;
END_SET
END_PROPERTY

(*!
<summary>Provides the concrete type name used in diagnostics.</summary>
<description>
Returns borrowed read-only metadata; keep the instance alive and do not modify the referenced string.
Initialized static storage is ready during base Task.FB_init; this getter has no side effects or exceptions.
</description>
*)
{attribute 'monitoring' := 'call'}
PROPERTY ClassName : REFERENCE TO STRING
GET
ClassName REF= _ClassName;
END_GET
END_PROPERTY

(*!
<summary>Provides the configured path for the file operation.</summary>
<description>
The setter copies text without performing I/O. Configure before Start and keep unchanged until STOPPED; Reset
preserves it. The native service determines whether the path is usable.
</description>
*)
{attribute 'monitoring' := 'call'}
PROPERTY FilePath : Tc2_System.T_MaxString
GET
FilePath := _LoadFile.sPathName;
END_GET
SET
_LoadFile.sPathName := FilePath;
END_SET
END_PROPERTY

(*!
<summary>Reports the byte count from a successfully completed load.</summary>
<description>
Returns the native result only while State.Stopped and FinalStopReason.WorkDone are both TRUE. In every other
state, including READY, RUNNING, failure and cancellation, returns the initial value of the property type.
This default is not a success indicator; inspect the task state and final reason. Zero outside successful
completion does not mean the target buffer was unchanged. The getter does not modify native outputs or
buffers. Copy a successful result before Reset or reuse.
</description>
*)
{attribute 'monitoring' := 'call'}
PROPERTY LoadedBytesCount : UDINT
GET
IF NOT State.Stopped OR_ELSE NOT FinalStopReason.WorkDone THEN
	RETURN;
END_IF

LoadedBytesCount := _LoadFile.cbRead;
END_GET
END_PROPERTY

(*!
<summary>Provides the library namespace used in diagnostics.</summary>
<description>Returns borrowed read-only namespace storage; do not modify the referenced string.</description>
*)
{attribute 'monitoring' := 'call'}
PROPERTY NamespaceName : REFERENCE TO STRING
GET
NamespaceName REF= CurrentNamespace.Name;
END_GET
END_PROPERTY

(*!
<summary>Resets the native request edge after the task has stopped.</summary>
<description>
Preserves configured inputs and does not undo completed filesystem effects. Pending I/O must finish during
stopping before this hook runs.
</description>
*)
METHOD PROTECTED OnReset
_LoadFile(bExecute := FALSE);
END_METHOD

(*!
<summary>Submits and advances a native file load into caller-owned memory.</summary>
<description>
Validates required configuration before submitting the request. Native errors raise an exception for the base
Task failure/stopping path without dynamic string-builder allocations. Normal completion reports DONE only
after the native block is no longer busy. No rollback is performed.
</description>
<param name="processingState">BUSY while pending; DONE after native completion without an error.</param>
<param name="stopReasonMessage">Not changed here; failures are passed through exceptions.</param>
*)
METHOD PROTECTED OnRunning
VAR_OUTPUT
	processingState : TOF_Tasks.TASK_PROCESSING_STATE;
END_VAR
VAR_IN_OUT
	stopReasonMessage : TOF_Core.ERROR_MESSAGE;
END_VAR
VAR
	formattedExceptionMessage : TOF_Core.ERROR_MESSAGE;
END_VAR
IF NOT _LoadFile.bExecute THEN 
	IF TOF_Core.Strings.IsNullOrWhiteSpace(stringToCheck := _LoadFile.sPathName) THEN
		TOF_Core.Exceptions.ThrowDataMemberNotSpecified(
			sourceNamespaceName := NamespaceName,
			sourceClassName := ClassName,
			sourcePOUName := __POUNAME(),
			sourcePosition := __POSITION(),
			dataMemberName := 'FilePath'
		);		
	END_IF

	IF _LoadFile.pReadBuff = 0 THEN
		TOF_Core.Exceptions.ThrowDataMemberNotSpecified(
			sourceNamespaceName := NamespaceName,
			sourceClassName := ClassName,
			sourcePOUName := __POUNAME(),
			sourcePosition := __POSITION(),
			dataMemberName := 'TargetBuffer'
		);		
	END_IF

	IF _LoadFile.cbReadLen = 0 THEN
		TOF_Core.Exceptions.ThrowDataMemberNotSpecified(
			sourceNamespaceName := NamespaceName,
			sourceClassName := ClassName,
			sourcePOUName := __POUNAME(),
			sourcePosition := __POSITION(),
			dataMemberName := 'TargetBufferSize'
		);		
	END_IF
END_IF

_LoadFile(bExecute := TRUE);

IF _LoadFile.bError THEN
	TOF_Core.WideStrings.Append255(
		formattedExceptionMessage,
		"An error occurred while loading the file '",
		TO_WSTRING(_LoadFile.sPathName),
		"'");

	FileSystemExceptions.ThrowFileSystem(
		sourceNamespaceName := NamespaceName,
		sourceClassName := ClassName,
		sourcePOUName := __POUNAME(),
		sourcePosition := __POSITION(),
		message := formattedExceptionMessage,
		errorCode := _LoadFile.nErrId
	);
END_IF

IF NOT _LoadFile.bBusy THEN
	processingState := TOF_Tasks.TASK_PROCESSING_STATE.DONE;
END_IF
END_METHOD

(*!
<summary>Waits for an already submitted operation before task termination.</summary>
<description>
Runs for every stop reason. Advances the pending FB with bExecute=FALSE without issuing another request.
Completion does not roll back side effects. Keep configuration and borrowed buffers valid until STOPPED.
</description>
<param name="readyToRelease">TRUE when the underlying FB is no longer busy.</param>
*)
METHOD PROTECTED OnStopping
VAR_OUTPUT
	readyToRelease : BOOL;
END_VAR
IF _LoadFile.bBusy THEN
	_LoadFile(bExecute := FALSE);
END_IF

readyToRelease := NOT _LoadFile.bBusy;
END_METHOD

(*!
<summary>Reports the size of this concrete instance in bytes.</summary>
*)
{attribute 'monitoring' := 'call'}
PROPERTY SelfSize : ULINT
GET
SelfSize := XSIZEOF(THIS^);
END_GET
END_PROPERTY

(*!
<summary>Specifies the caller-owned writable buffer for loading file bytes.</summary>
<description>
Provide at least TargetBufferSize bytes and retain the buffer until STOPPED, including after cancellation or
failure. Null is rejected during execution. The wrapper cannot validate actual capacity or lifetime. Do not
access the buffer concurrently. Failure does not restore previous contents.
</description>
*)
{attribute 'monitoring' := 'call'}
PROPERTY TargetBuffer : POINTER TO BYTE
GET
TargetBuffer := _LoadFile.pReadBuff;
END_GET
SET
_LoadFile.pReadBuff := TargetBuffer;
END_SET
END_PROPERTY

(*!
<summary>Specifies the positive number of bytes requested from the file.</summary>
<description>
Passed to native cbReadLen. Must not exceed the caller-owned TargetBuffer capacity. Zero is rejected during
execution and identifies TargetBufferSize in the failure diagnostic. Keep this value unchanged from Start
through STOPPED. LoadedBytesCount reports the actual count only after successful completion; this setting does not assert that the entire file fits in the buffer.
</description>
*)
{attribute 'monitoring' := 'call'}
PROPERTY TargetBufferSize : UDINT
GET
TargetBufferSize := _LoadFile.cbReadLen;
END_GET
SET
_LoadFile.cbReadLen := TargetBufferSize;
END_SET
END_PROPERTY

(*!
<summary>Configures the timeout passed to native operation requests.</summary>
<description>
Set before Start and keep unchanged until STOPPED. Reset preserves this value. It is not an overall task
deadline or a guarantee of resource release after a timeout.
</description>
*)
{attribute 'monitoring' := 'call'}
PROPERTY Timeout : TIME
GET
Timeout := _LoadFile.tTimeout;
END_GET
SET
_LoadFile.tTimeout := Timeout;
END_SET
END_PROPERTY

END_FUNCTION_BLOCK

// ---- Tasks/File/RenameFile.TcPOU
(*
SPDX-FileCopyrightText: © 2026 Oleksandr Tiutyk <trofimich@gmail.com>
SPDX-License-Identifier: MIT
License: https://opensource.org/license/mit
*)

(*!
<summary>Renames a file through cyclic task execution.</summary>
<description>
Use one owner task. Configure both paths, target, path type and timeout before Start and keep them unchanged
until STOPPED. Both paths are required during execution. The native service determines path and destination
collision behavior; this wrapper adds no overwrite, retry or rollback policy and reports native errors through
Task failure handling. Continue Execute through stopping after cancellation; pending native work must finish.
Failure or cancellation does not prove the original names were preserved. Reset preserves configuration.
</description>
*)

{attribute 'no_explicit_call' := 'do not call this function block directly'}
FUNCTION_BLOCK RenameFile EXTENDS TOF_Tasks.Task IMPLEMENTS IFileSystemTask
VAR_STAT
	//! <summary>Static type metadata available before the base task initializes its default name.</summary>
	{attribute 'hide'}
	_ClassName : STRING := __POUNAME();
END_VAR
VAR
    _RenameFile : Tc2_System.FB_FileRename;
END_VAR

(*!
<summary>Selects the ADS target for the native filesystem operation.</summary>
<description>
Configure before Start and keep unchanged until STOPPED; the setter stores configuration without submitting
I/O.
</description>
*)
{attribute 'monitoring' := 'call'}
{attribute 'OPC.UA.DA.Property' := '1'}
{attribute 'OPC.UA.DA' := '1'}
PROPERTY AmsNetId : Tc2_System.T_AmsNetID
GET
AmsNetId := _RenameFile.sNetId;
END_GET
SET
_RenameFile.sNetId := AmsNetId;
END_SET
END_PROPERTY

(*!
<summary>Provides the concrete type name used in diagnostics.</summary>
<description>
Returns borrowed read-only metadata; keep the instance alive and do not modify the referenced string.
Initialized static storage is ready during base Task.FB_init; this getter has no side effects or exceptions.
</description>
*)
{attribute 'monitoring' := 'call'}
PROPERTY ClassName : REFERENCE TO STRING
GET
ClassName REF= _ClassName;
END_GET
END_PROPERTY

(*!
<summary>Provides the library namespace used in diagnostics.</summary>
<description>Returns borrowed read-only namespace storage; do not modify the referenced string.</description>
*)
{attribute 'monitoring' := 'call'}
PROPERTY NamespaceName : REFERENCE TO STRING
GET
NamespaceName REF= CurrentNamespace.Name;
END_GET
END_PROPERTY

(*!
<summary>Provides the requested destination path for the rename operation.</summary>
<description>
Configure before Start and keep unchanged until STOPPED. Assignment does not reserve the destination or
guarantee replacement of an existing entry. Native collision behavior applies; Reset preserves it.
</description>
*)
{attribute 'monitoring' := 'call'}
{attribute 'OPC.UA.DA.Property' := '1'}
{attribute 'OPC.UA.DA' := '1'}
PROPERTY NewFilePath : Tc2_System.T_MaxString
GET
NewFilePath := _RenameFile.sNewName;
END_GET
SET
_RenameFile.sNewName := NewFilePath;
END_SET
END_PROPERTY

(*!
<summary>Provides the source path for the rename operation.</summary>
<description>
Configure before Start and keep unchanged until STOPPED. The setter copies text; native execution checks the
source. Reset preserves it.
</description>
*)
{attribute 'monitoring' := 'call'}
{attribute 'OPC.UA.DA.Property' := '1'}
{attribute 'OPC.UA.DA' := '1'}
PROPERTY OldFilePath : Tc2_System.T_MaxString
GET
OldFilePath := _RenameFile.sOldName;
END_GET
SET
_RenameFile.sOldName := OldFilePath;
END_SET
END_PROPERTY

(*!
<summary>Resets the native request edge after the task has stopped.</summary>
<description>
Preserves configured inputs and does not undo completed filesystem effects. Pending I/O must finish during
stopping before this hook runs.
</description>
*)
METHOD PROTECTED OnReset
_RenameFile(bExecute := FALSE);
END_METHOD

(*!
<summary>Submits and advances native renaming of the configured file.</summary>
<description>
Validates required configuration before submitting the request. Native errors raise an exception for the base
Task failure/stopping path without dynamic string-builder allocations. Normal completion reports DONE only
after the native block is no longer busy. No rollback is performed.
</description>
<param name="processingState">BUSY while pending; DONE after native completion without an error.</param>
<param name="stopReasonMessage">Not changed here; failures are passed through exceptions.</param>
*)
METHOD PROTECTED OnRunning
VAR_OUTPUT
	processingState : TOF_Tasks.TASK_PROCESSING_STATE;
END_VAR
VAR_IN_OUT
	stopReasonMessage : TOF_Core.ERROR_MESSAGE;
END_VAR
VAR
	formattedExceptionMessage : TOF_Core.ERROR_MESSAGE;
END_VAR
IF NOT _RenameFile.bExecute THEN 
	IF TOF_Core.Strings.IsNullOrWhiteSpace(stringToCheck := _RenameFile.sOldName) THEN
		TOF_Core.Exceptions.ThrowDataMemberNotSpecified(
			sourceNamespaceName := NamespaceName,
			sourceClassName := ClassName,
			sourcePOUName := __POUNAME(),
			sourcePosition := __POSITION(),
			dataMemberName := 'OldFilePath'
		);		
	END_IF

	IF TOF_Core.Strings.IsNullOrWhiteSpace(stringToCheck := _RenameFile.sNewName) THEN
		TOF_Core.Exceptions.ThrowDataMemberNotSpecified(
			sourceNamespaceName := NamespaceName,
			sourceClassName := ClassName,
			sourcePOUName := __POUNAME(),
			sourcePosition := __POSITION(),
			dataMemberName := 'NewFilePath'
		);		
	END_IF
	
	_RenameFile(bExecute := FALSE);
END_IF

_RenameFile(bExecute := TRUE);

IF _RenameFile.bError THEN
	TOF_Core.WideStrings.Append255(
		formattedExceptionMessage,
		"An error occurred while renaming the file '",
		TO_WSTRING(_RenameFile.sOldName),
		"' to '",
		TO_WSTRING(_RenameFile.sNewName),
		"'");

	FileSystemExceptions.ThrowFileSystem(
		sourceNamespaceName := NamespaceName,
		sourceClassName := ClassName,
		sourcePOUName := __POUNAME(),
		sourcePosition := __POSITION(),
		message := formattedExceptionMessage,
		errorCode := _RenameFile.nErrId
	);
END_IF

IF NOT _RenameFile.bBusy THEN
	processingState := TOF_Tasks.TASK_PROCESSING_STATE.DONE;
END_IF
END_METHOD

(*!
<summary>Waits for an already submitted operation before task termination.</summary>
<description>
Runs for every stop reason. Advances the pending FB with bExecute=FALSE without issuing another request.
Completion does not roll back side effects. Keep configuration and borrowed buffers valid until STOPPED.
</description>
<param name="readyToRelease">TRUE when the underlying FB is no longer busy.</param>
*)
METHOD PROTECTED OnStopping
VAR_OUTPUT
	readyToRelease : BOOL;
END_VAR
IF _RenameFile.bBusy THEN
	_RenameFile(bExecute := FALSE);
END_IF

readyToRelease := NOT _RenameFile.bBusy;
END_METHOD

(*!
<summary>Selects the native path context for the filesystem request.</summary>
<description>
Configure before Start and keep unchanged until STOPPED. It is passed to the native operation, not used as a
path-validity result. Reset preserves it.
</description>
*)
{attribute 'monitoring' := 'call'}
{attribute 'OPC.UA.DA.Property' := '1'}
{attribute 'OPC.UA.DA' := '1'}
PROPERTY PathType : Tc2_System.E_OpenPath
GET
PathType := _RenameFile.ePath;
END_GET
SET
_RenameFile.ePath := PathType;
END_SET
END_PROPERTY

(*!
<summary>Reports the size of this concrete instance in bytes.</summary>
*)
{attribute 'monitoring' := 'call'}
PROPERTY SelfSize : ULINT
GET
SelfSize := XSIZEOF(THIS^);
END_GET
END_PROPERTY

(*!
<summary>Configures the timeout passed to native operation requests.</summary>
<description>
Set before Start and keep unchanged until STOPPED. Reset preserves this value. It is not an overall task
deadline or a guarantee of resource release after a timeout.
</description>
*)
{attribute 'monitoring' := 'call'}
{attribute 'OPC.UA.DA.Property' := '1'}
{attribute 'OPC.UA.DA' := '1'}
PROPERTY Timeout : TIME
GET
Timeout := _RenameFile.tTimeout;
END_GET
SET
_RenameFile.tTimeout := Timeout;
END_SET
END_PROPERTY

END_FUNCTION_BLOCK
